Universal Robots PolyScope program: PasteExtrusion.urp

Program PasteExtrusion (installation=GCode_CeramicPaste directory=/programs createdIn=5.11.5.1010327 lastSavedIn=5.11.5.1010327 robotSerialNumber=20205000256)
Calibrated DH parameters: a=[-0.00012, -0.537495, -0.054766, -0.000072, -0.000096, 0]; d=[0.180617, 85.726709, 533.143122, -618.695874, 0.119802, 0.115691]; alpha=[1.570127, -0.003428, -0.000919, 1.569861, -1.571555, 0]; deltaTheta=[0, -0.500372, 5.308769, 1.474786, -0.000002, 0]
BeforeStart
  Set DigitalOutput pin=Speed_b0; digitalValue=0
  Set DigitalOutput pin=Speed_b1; digitalValue=0
  Set DigitalOutput pin=digital_out[2]; digitalValue=0
  Set DigitalOutput pin=digital_out[3]; digitalValue=0
  Set DigitalOutput pin=tool_out[0]; digitalValue=0
  Set DigitalOutput pin=tool_out[1]; digitalValue=0
Robot Program (runOnlyOnce=true)
  Popup Message (haltProgram=false message=Start print? inputType=Text)
  MoveL speed 250 mm/s, acceleration 1200 mm/s^2 (useActiveTCP=true) feature=Base
    Waypoint Waypoint (Variable): variable(featureName=Datum)
  URCap Toolpath Move (Remote TCP & Toolpath, Universal Robots A/S) dataModel(subtreeCreated=true, SELECTED_RTCP=TCP, TOOL_ACCELERATION=500.0, RTCP_COMMON_DATAMODEL_FREESPINZ=false)
    URCap Toolpath (Remote TCP & Toolpath, Universal Robots A/S) dataModel(WAYPOINT_NAME=Toolpath_1, SELECTED_PCS=Datum, WAYPOINT_TOOLACC=1000.0, RTCP_TOOLPATH_DATAMODEL_TOOLACCELERATIONSELECTION=SHARED, WAYPOINT_TOOLSPEED=100.0, RTCP_TOOLPATH_DATAMODEL_TOOLSPEEDSELECTION=FEEDRATE, TOOLPATH_NAME=run1.nc)
    URCap Toolpath (Remote TCP & Toolpath, Universal Robots A/S) dataModel(WAYPOINT_NAME=Toolpath_2, SELECTED_PCS=Datum, RTCP_TOOLPATH_DATAMODEL_TOOLSPEEDSELECTION=FEEDRATE, TOOLPATH_NAME=run2.nc)
    URCap Toolpath (Remote TCP & Toolpath, Universal Robots A/S) dataModel(WAYPOINT_NAME=Toolpath_3, SELECTED_PCS=Datum, RTCP_TOOLPATH_DATAMODEL_TOOLSPEEDSELECTION=FEEDRATE, TOOLPATH_NAME=run3.nc)
    URCap Toolpath (Remote TCP & Toolpath, Universal Robots A/S) dataModel(WAYPOINT_NAME=Toolpath_4, SELECTED_PCS=Datum, RTCP_TOOLPATH_DATAMODEL_TOOLSPEEDSELECTION=FEEDRATE, TOOLPATH_NAME=run4.nc)
    URCap Toolpath (Remote TCP & Toolpath, Universal Robots A/S) dataModel(WAYPOINT_NAME=Toolpath_5, SELECTED_PCS=Datum, RTCP_TOOLPATH_DATAMODEL_TOOLSPEEDSELECTION=FEEDRATE, TOOLPATH_NAME=run5.nc)
  Set DigitalOutput pin=Speed_b0; digitalValue=0
  Set DigitalOutput pin=Speed_b1; digitalValue=0
  Set DigitalOutput pin=digital_out[2]; digitalValue=0
  Set DigitalOutput pin=digital_out[3]; digitalValue=0
Thread Thread_1 (runOnlyOnce=false)
  If ResetFlow0
    Set AnalogOutput pin=analog_out[0]; analogValue=1
    Set DigitalOutput pin=tool_out[0]; digitalValue=0
  If ResetFlow1
    Set AnalogOutput pin=analog_out[1]; analogValue=1
    Set DigitalOutput pin=tool_out[1]; digitalValue=0
  Script: sync()
